TEXTLIST TL_E_CTRL_XPU
  0 = 'XTS_CMD_NULL'
  10 = 'XTS_CMD_INIT'
  30 = 'XTS_IDLE'
   = ''
END_TEXTLIST

(* stored: Version 1.1.0.1
   TextList TL_E_CTRL_XPU: Id {62ee145b-05f5-4a19-9535-b86c8df68e2e} *)
